FUNCTION_BLOCK ControlTS (* Composite Function Block Type *)
  (* Standard: 61499-2 *)
  (* Version 0.0, 6/3/2016, Andrei, nxtControl GmbH, template *)
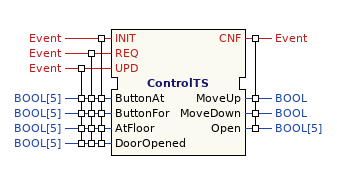
  EVENT_INPUT
    INIT WITH AtFloor, DoorOpened, ButtonAt, ButtonFor; (* Initialization Request *)
    REQ WITH ButtonAt, ButtonFor, AtFloor, DoorOpened; (* Normal Execution Request *)
    UPD WITH AtFloor, DoorOpened, ButtonFor, ButtonAt;
  END_EVENT
  EVENT_OUTPUT
    CNF WITH MoveUp, MoveDown, Open; (* Execution Confirmation *)
  END_EVENT
  VAR_INPUT
    ButtonAt : ARRAY [0..4] OF BOOL;
    ButtonFor : ARRAY [0..4] OF BOOL;
    AtFloor : ARRAY [0..4] OF BOOL; (* Input event qualifier *)
    DoorOpened : ARRAY [0..4] OF BOOL;
  END_VAR
  VAR_OUTPUT
    MoveUp : BOOL; (* Output event qualifier *)
    MoveDown : BOOL;
    Open : ARRAY [0..4] OF BOOL;
  END_VAR
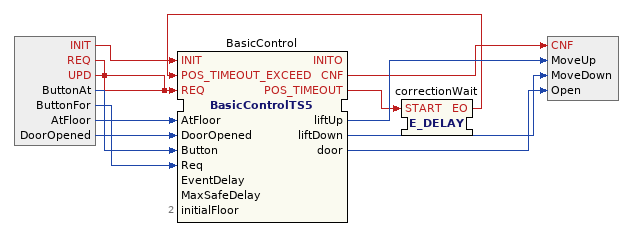
  FBS
    correctionWait : E_DELAY;
    BasicControl : BasicControlTS5(initialFloor := 2);
  END_FBS
  EVENT_CONNECTIONS
    INIT TO BasicControl.INIT;
    REQ TO BasicControl.REQ;
    UPD TO BasicControl.REQ;
    correctionWait.EO TO BasicControl.POS_TIMEOUT_EXCEED;
    BasicControl.CNF TO CNF;
    BasicControl.POS_TIMEOUT TO correctionWait.START;
  END_CONNECTIONS
  DATA_CONNECTIONS
    AtFloor TO BasicControl.AtFloor;
    DoorOpened TO BasicControl.DoorOpened;
    ButtonAt TO BasicControl.Button;
    ButtonFor TO BasicControl.Req;
    BasicControl.liftUp TO MoveUp;
    BasicControl.liftDown TO MoveDown;
    BasicControl.door TO Open;
  END_CONNECTIONS
END_FUNCTION_BLOCK
